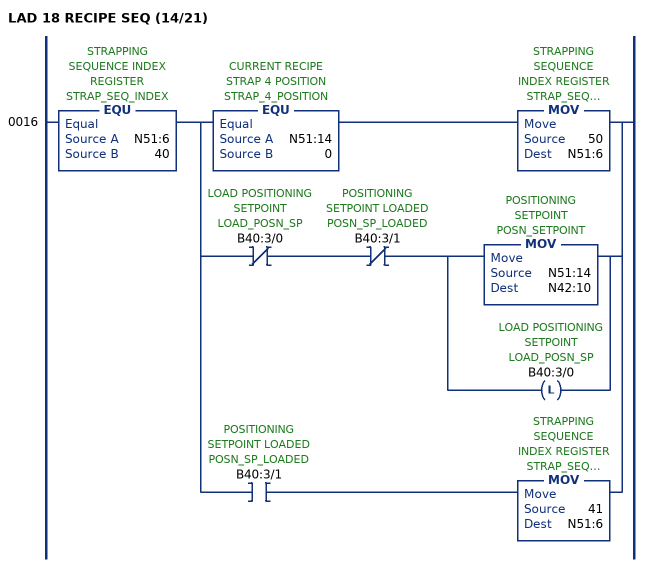
% Rung: 16 %
SOR EQU N51:6 40 BST EQU N51:14 0 MOV 50 N51:6 NXB XIO B40:3/0 XIO B40:3/1 BST MOV N51:14 N42:10 NXB OTL B40:3/0 BND NXB XIC B40:3/1 MOV 41 N51:6 BND EOR
%   N51:6  STRAP_SEQ_INDEX  "STRAPPING SEQUENCE INDEX REGISTER" %
%   N51:14  STRAP_4_POSITION  "CURRENT RECIPE STRAP 4 POSITION" %
%   B40:3/0  LOAD_POSN_SP  "LOAD POSITIONING SETPOINT" %
%   B40:3/1  POSN_SP_LOADED  "POSITIONING SETPOINT LOADED" %
%   N42:10  POSN_SETPOINT  "POSITIONING SETPOINT" %

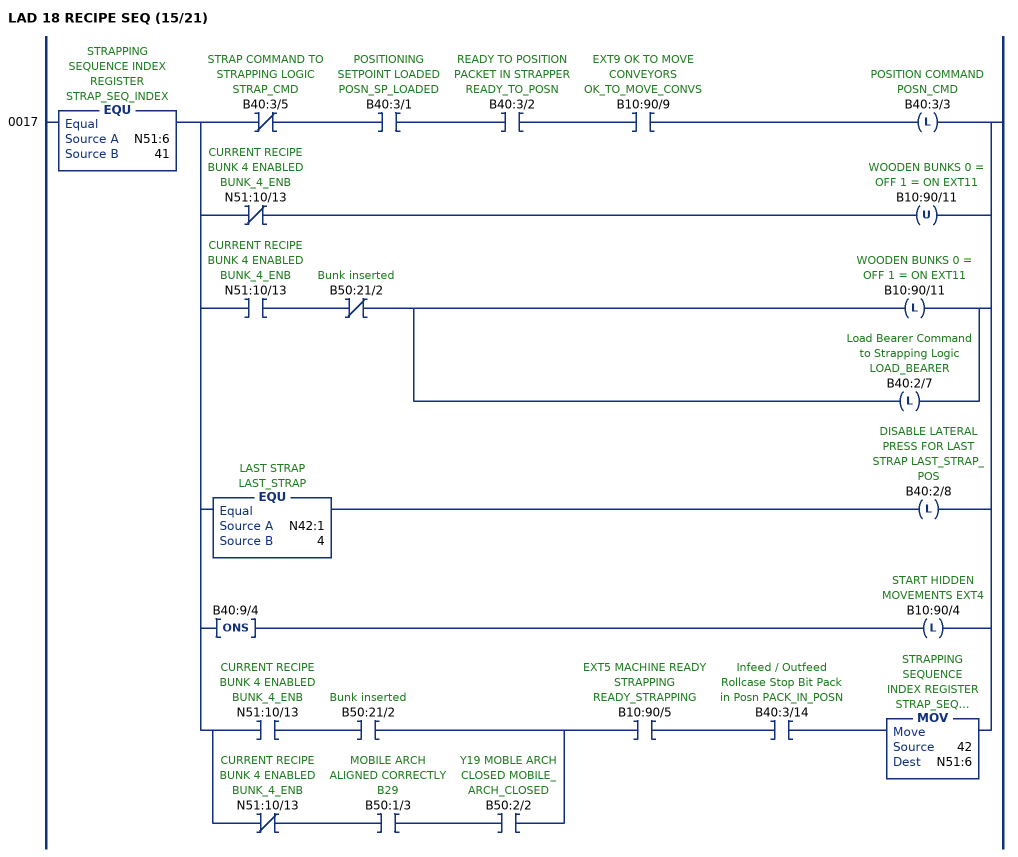
% Rung: 17 %
SOR EQU N51:6 41 BST XIO B40:3/5 XIC B40:3/1 XIC B40:3/2 XIC B10:90/9 OTL B40:3/3 NXB XIO N51:10/13 OTU B10:90/11 NXB XIC N51:10/13 XIO B50:21/2 BST OTL B10:90/11 NXB OTL B40:2/7 BND NXB EQU N42:1 4 OTL B40:2/8 NXB ONS B40:9/4 OTL B10:90/4 NXB BST XIC N51:10/13 XIC B50:21/2 NXB XIO N51:10/13 XIC B50:1/3 XIC B50:2/2 BND XIC B10:90/5 XIC B40:3/14 MOV 42 N51:6 BND EOR
%   N51:6  STRAP_SEQ_INDEX  "STRAPPING SEQUENCE INDEX REGISTER" %
%   B40:3/5  STRAP_CMD  "STRAP COMMAND TO STRAPPING LOGIC" %
%   B40:3/1  POSN_SP_LOADED  "POSITIONING SETPOINT LOADED" %
%   B40:3/2  READY_TO_POSN  "READY TO POSITION PACKET IN STRAPPER" %
%   B10:90/9  OK_TO_MOVE_CONVS  "EXT9 OK TO MOVE CONVEYORS" %
%   B40:3/3  POSN_CMD  "POSITION COMMAND" %
%   N51:10/13  BUNK_4_ENB  "CURRENT RECIPE BUNK 4 ENABLED" %
%   B10:90/11  EXT11  "WOODEN BUNKS 0 = OFF 1 = ON" %
%   B50:21/2  "Bunk inserted" %
%   B40:2/7  LOAD_BEARER  "Load Bearer Command to Strapping Logic" %
%   N42:1  LAST_STRAP  "LAST STRAP" %
%   B40:2/8  LAST_STRAP_POS  "DISABLE LATERAL PRESS FOR LAST STRAP" %
%   B10:90/4  EXT4  "START HIDDEN MOVEMENTS" %
%   B50:1/3  B29  "MOBILE ARCH ALIGNED CORRECTLY" %
%   B50:2/2  MOBILE_ARCH_CLOSED  "Y19 MOBLE ARCH CLOSED" %
%   B10:90/5  READY_STRAPPING  "EXT5 MACHINE READY STRAPPING" %
%   B40:3/14  PACK_IN_POSN  "Infeed / Outfeed Rollcase Stop Bit Pack in Posn" %

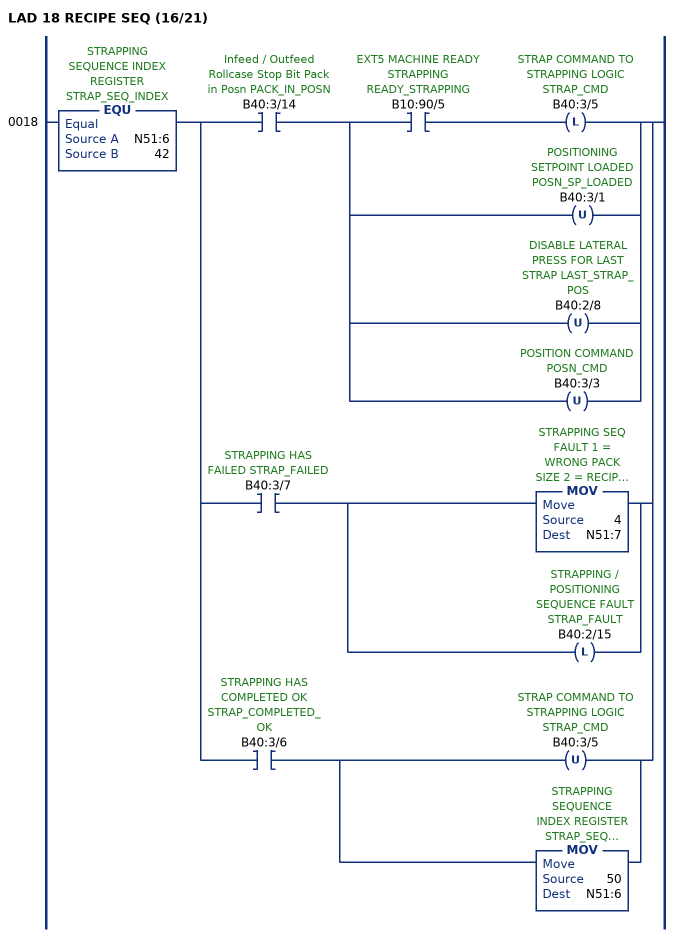
% Rung: 18 %
SOR EQU N51:6 42 BST XIC B40:3/14 BST XIC B10:90/5 OTL B40:3/5 NXB OTU B40:3/1 NXB OTU B40:2/8 NXB OTU B40:3/3 BND NXB XIC B40:3/7 BST MOV 4 N51:7 NXB OTL B40:2/15 BND NXB XIC B40:3/6 BST OTU B40:3/5 NXB MOV 50 N51:6 BND BND EOR
%   N51:6  STRAP_SEQ_INDEX  "STRAPPING SEQUENCE INDEX REGISTER" %
%   B40:3/14  PACK_IN_POSN  "Infeed / Outfeed Rollcase Stop Bit Pack in Posn" %
%   B10:90/5  READY_STRAPPING  "EXT5 MACHINE READY STRAPPING" %
%   B40:3/5  STRAP_CMD  "STRAP COMMAND TO STRAPPING LOGIC" %
%   B40:3/1  POSN_SP_LOADED  "POSITIONING SETPOINT LOADED" %
%   B40:2/8  LAST_STRAP_POS  "DISABLE LATERAL PRESS FOR LAST STRAP" %
%   B40:3/3  POSN_CMD  "POSITION COMMAND" %
%   B40:3/7  STRAP_FAILED  "STRAPPING HAS FAILED" %
%   N51:7  STRAP_SEQ_FLT  "STRAPPING SEQ FAULT 1 = WRONG PACK SIZE 2 = RECIPE FAULT 3 = POSNING FAULT 4 = STRAPPING FAULT" %
%   B40:2/15  STRAP_FAULT  "STRAPPING / POSITIONING SEQUENCE FAULT" %
%   B40:3/6  STRAP_COMPLETED_OK  "STRAPPING HAS COMPLETED OK" %

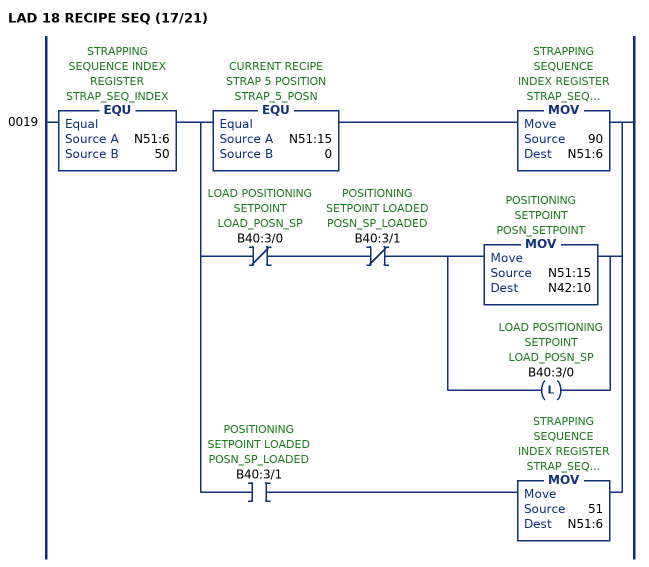
% Rung: 19 %
SOR EQU N51:6 50 BST EQU N51:15 0 MOV 90 N51:6 NXB XIO B40:3/0 XIO B40:3/1 BST MOV N51:15 N42:10 NXB OTL B40:3/0 BND NXB XIC B40:3/1 MOV 51 N51:6 BND EOR
%   N51:6  STRAP_SEQ_INDEX  "STRAPPING SEQUENCE INDEX REGISTER" %
%   N51:15  STRAP_5_POSN  "CURRENT RECIPE STRAP 5 POSITION" %
%   B40:3/0  LOAD_POSN_SP  "LOAD POSITIONING SETPOINT" %
%   B40:3/1  POSN_SP_LOADED  "POSITIONING SETPOINT LOADED" %
%   N42:10  POSN_SETPOINT  "POSITIONING SETPOINT" %

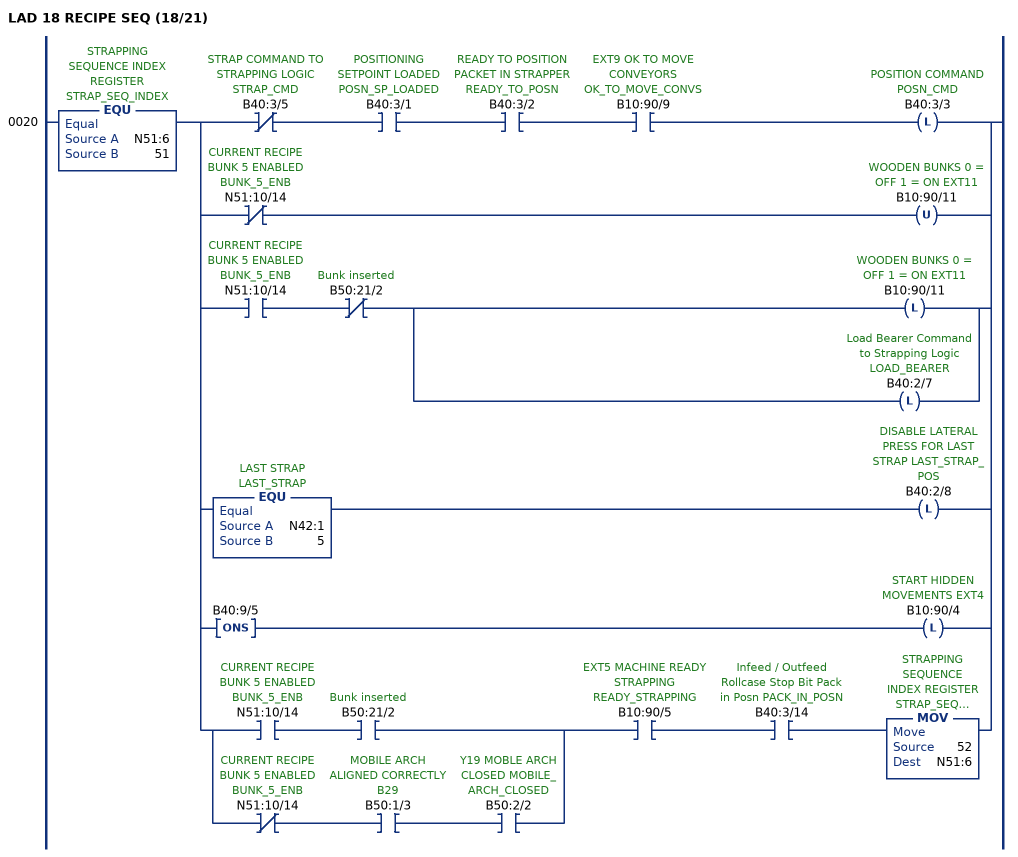
% Rung: 20 %
SOR EQU N51:6 51 BST XIO B40:3/5 XIC B40:3/1 XIC B40:3/2 XIC B10:90/9 OTL B40:3/3 NXB XIO N51:10/14 OTU B10:90/11 NXB XIC N51:10/14 XIO B50:21/2 BST OTL B10:90/11 NXB OTL B40:2/7 BND NXB EQU N42:1 5 OTL B40:2/8 NXB ONS B40:9/5 OTL B10:90/4 NXB BST XIC N51:10/14 XIC B50:21/2 NXB XIO N51:10/14 XIC B50:1/3 XIC B50:2/2 BND XIC B10:90/5 XIC B40:3/14 MOV 52 N51:6 BND EOR
%   N51:6  STRAP_SEQ_INDEX  "STRAPPING SEQUENCE INDEX REGISTER" %
%   B40:3/5  STRAP_CMD  "STRAP COMMAND TO STRAPPING LOGIC" %
%   B40:3/1  POSN_SP_LOADED  "POSITIONING SETPOINT LOADED" %
%   B40:3/2  READY_TO_POSN  "READY TO POSITION PACKET IN STRAPPER" %
%   B10:90/9  OK_TO_MOVE_CONVS  "EXT9 OK TO MOVE CONVEYORS" %
%   B40:3/3  POSN_CMD  "POSITION COMMAND" %
%   N51:10/14  BUNK_5_ENB  "CURRENT RECIPE BUNK 5 ENABLED" %
%   B10:90/11  EXT11  "WOODEN BUNKS 0 = OFF 1 = ON" %
%   B50:21/2  "Bunk inserted" %
%   B40:2/7  LOAD_BEARER  "Load Bearer Command to Strapping Logic" %
%   N42:1  LAST_STRAP  "LAST STRAP" %
%   B40:2/8  LAST_STRAP_POS  "DISABLE LATERAL PRESS FOR LAST STRAP" %
%   B10:90/4  EXT4  "START HIDDEN MOVEMENTS" %
%   B50:1/3  B29  "MOBILE ARCH ALIGNED CORRECTLY" %
%   B50:2/2  MOBILE_ARCH_CLOSED  "Y19 MOBLE ARCH CLOSED" %
%   B10:90/5  READY_STRAPPING  "EXT5 MACHINE READY STRAPPING" %
%   B40:3/14  PACK_IN_POSN  "Infeed / Outfeed Rollcase Stop Bit Pack in Posn" %

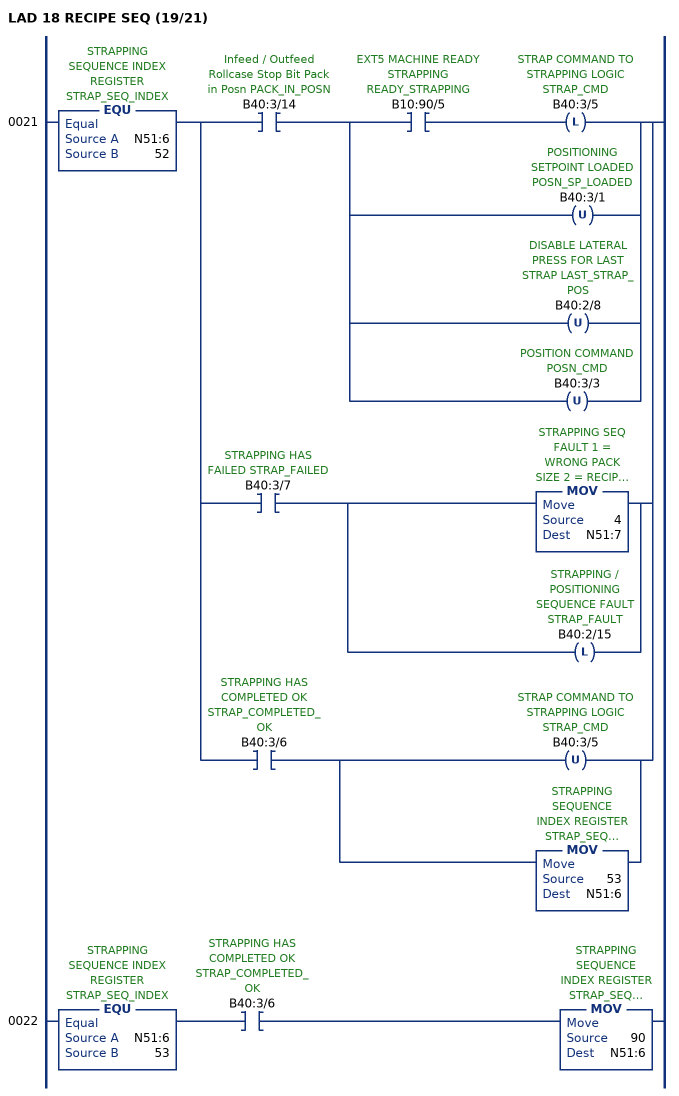
% Rung: 21 %
SOR EQU N51:6 52 BST XIC B40:3/14 BST XIC B10:90/5 OTL B40:3/5 NXB OTU B40:3/1 NXB OTU B40:2/8 NXB OTU B40:3/3 BND NXB XIC B40:3/7 BST MOV 4 N51:7 NXB OTL B40:2/15 BND NXB XIC B40:3/6 BST OTU B40:3/5 NXB MOV 53 N51:6 BND BND EOR
%   N51:6  STRAP_SEQ_INDEX  "STRAPPING SEQUENCE INDEX REGISTER" %
%   B40:3/14  PACK_IN_POSN  "Infeed / Outfeed Rollcase Stop Bit Pack in Posn" %
%   B10:90/5  READY_STRAPPING  "EXT5 MACHINE READY STRAPPING" %
%   B40:3/5  STRAP_CMD  "STRAP COMMAND TO STRAPPING LOGIC" %
%   B40:3/1  POSN_SP_LOADED  "POSITIONING SETPOINT LOADED" %
%   B40:2/8  LAST_STRAP_POS  "DISABLE LATERAL PRESS FOR LAST STRAP" %
%   B40:3/3  POSN_CMD  "POSITION COMMAND" %
%   B40:3/7  STRAP_FAILED  "STRAPPING HAS FAILED" %
%   N51:7  STRAP_SEQ_FLT  "STRAPPING SEQ FAULT 1 = WRONG PACK SIZE 2 = RECIPE FAULT 3 = POSNING FAULT 4 = STRAPPING FAULT" %
%   B40:2/15  STRAP_FAULT  "STRAPPING / POSITIONING SEQUENCE FAULT" %
%   B40:3/6  STRAP_COMPLETED_OK  "STRAPPING HAS COMPLETED OK" %
% Rung: 22 %
SOR EQU N51:6 53 XIC B40:3/6 MOV 90 N51:6 EOR
%   N51:6  STRAP_SEQ_INDEX  "STRAPPING SEQUENCE INDEX REGISTER" %
%   B40:3/6  STRAP_COMPLETED_OK  "STRAPPING HAS COMPLETED OK" %

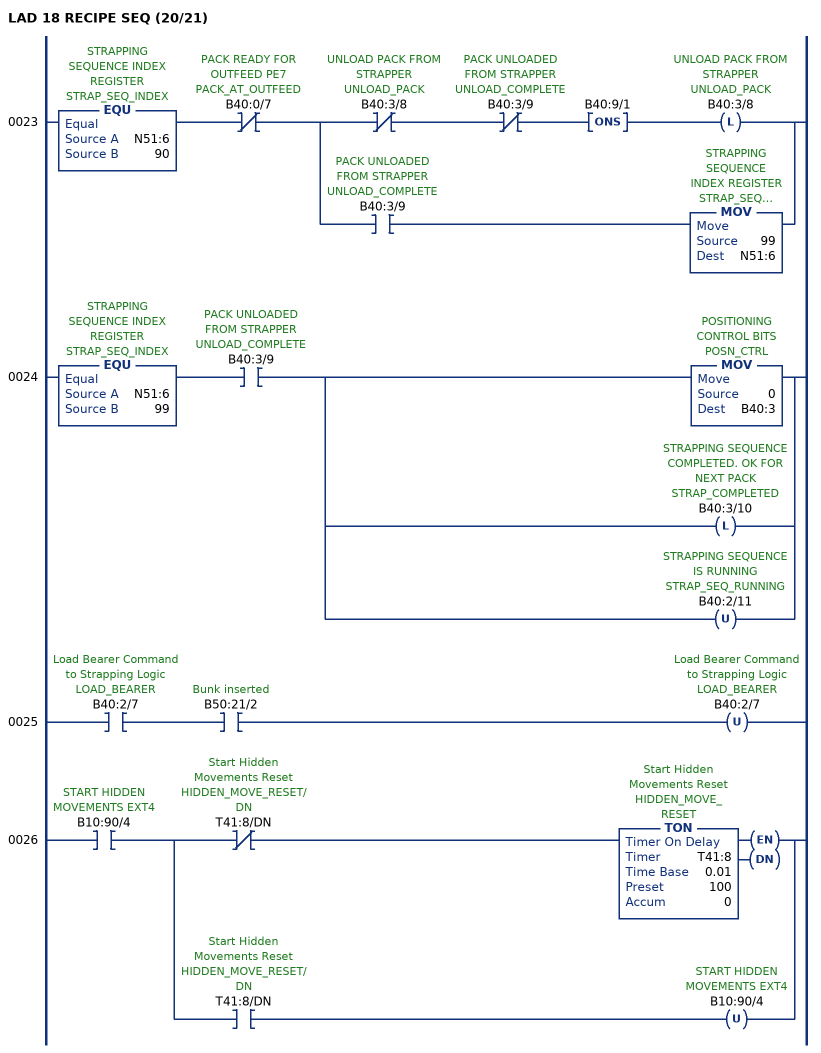
% Rung: 23 %
SOR EQU N51:6 90 XIO B40:0/7 BST XIO B40:3/8 XIO B40:3/9 ONS B40:9/1 OTL B40:3/8 NXB XIC B40:3/9 MOV 99 N51:6 BND EOR
%   N51:6  STRAP_SEQ_INDEX  "STRAPPING SEQUENCE INDEX REGISTER" %
%   B40:0/7  PACK_AT_OUTFEED  "PACK READY FOR OUTFEED PE7" %
%   B40:3/8  UNLOAD_PACK  "UNLOAD PACK FROM STRAPPER" %
%   B40:3/9  UNLOAD_COMPLETE  "PACK UNLOADED FROM STRAPPER" %
% Rung: 24 %
SOR EQU N51:6 99 XIC B40:3/9 BST MOV 0 B40:3 NXB OTL B40:3/10 NXB OTU B40:2/11 BND EOR
%   N51:6  STRAP_SEQ_INDEX  "STRAPPING SEQUENCE INDEX REGISTER" %
%   B40:3/9  UNLOAD_COMPLETE  "PACK UNLOADED FROM STRAPPER" %
%   B40:3  POSN_CTRL  "POSITIONING CONTROL BITS" %
%   B40:3/10  STRAP_COMPLETED  "STRAPPING SEQUENCE COMPLETED. OK FOR NEXT PACK" %
%   B40:2/11  STRAP_SEQ_RUNNING  "STRAPPING SEQUENCE IS RUNNING" %
% Rung: 25 %
SOR XIC B40:2/7 XIC B50:21/2 OTU B40:2/7 EOR
%   B40:2/7  LOAD_BEARER  "Load Bearer Command to Strapping Logic" %
%   B50:21/2  "Bunk inserted" %
% Rung: 26 %
SOR XIC B10:90/4 BST XIO T41:8/DN TON T41:8 0.01 100 0 NXB XIC T41:8/DN OTU B10:90/4 BND EOR
%   B10:90/4  EXT4  "START HIDDEN MOVEMENTS" %
%   T41:8  HIDDEN_MOVE_RESET  "Start Hidden Movements Reset" %

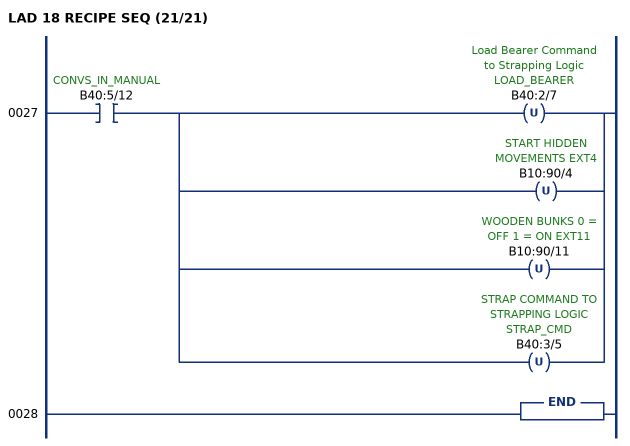
% Rung: 27 %
SOR XIC B40:5/12 BST OTU B40:2/7 NXB OTU B10:90/4 NXB OTU B10:90/11 NXB OTU B40:3/5 BND EOR
%   B40:5/12  CONVS_IN_MANUAL %
%   B40:2/7  LOAD_BEARER  "Load Bearer Command to Strapping Logic" %
%   B10:90/4  EXT4  "START HIDDEN MOVEMENTS" %
%   B10:90/11  EXT11  "WOODEN BUNKS 0 = OFF 1 = ON" %
%   B40:3/5  STRAP_CMD  "STRAP COMMAND TO STRAPPING LOGIC" %
% Rung: 28 %
SOR END EOR

OTHER DOCUMENTED ADDRESSES
  B1:0  "NOEM"
  B3:1/0  "Avl_Pres_vertical"
  B3:1/5  Y23  "Y23"
  B3:1/6  "Avl_Pres_lateral"
  B3:2/3  "IPWR"
  B3:2/4  "Par"
  B3:2/6  "Check_control_motor_ brake"
  B3:14/5  "High_pressure"
  B3:26  MPV  "MPV"
  B3:27  MPL  "MPL"
  B3:28  "FIX_FORCE_V_P"
  B3:29  I  "FIX_FORCE_L_P"
  B10:2/2  "H4"
  B10:2/3  "H5"
  B10:2/4  "EXT25"
  B10:2/5  "EXT26"
  B10:2/6  "EXT27"
  B10:2/7  "EXT28"
  B10:15/0  "OP_V_F_PRESS"
  B10:17/0  "Pack_Large"
  B10:18/0  "C_lpress_FIX_press"
  B10:19/0  "B_vpress_FIX_press"
  B10:33/5  F6  "F6-KEY"
  B10:90/0  "EXT0"
  B10:90/1  "EXT1"
  B10:90/2  "EXT2"
  B10:90/3  "EXT3"
  B10:90/7  "EXT7"
  B10:90/14  "EXT14"
  B10:90/15  "EXT15"
  B10:91/0  "EXT16"
  B10:91/1  "EXT17"
  B10:91/2  "EXT18"
  B10:91/3  "EXT19"
  B10:91/8  "EXT24"
  B10:100/6  "G_Corner"
  B10:100/7  "B_vpress_FIX_pres"
  B10:100/8  "C_lpress_FIX_pres"
  B10:100/9  "Pack_small"
  B20:0/2  "B3"
  B20:200/1  "E2"
  B40:0/12  PACK_STORAGE_PE_2  "Pack Index Point 3"
  B40:2/12  STRAP_SEQ_COMPLETE  "STRAPPING SEQUENCE IS COMPLETE"
  B40:3/4  PACK_POSNED  "PACK IS POSITIONED IN STRAPPER"
  B40:4  POSN_CTRL_2  "Position Control Bits Word 2"
  B40:4/6  LOAD_BEARER_PULSE  "Load Bearer Pulse To Strapping Logic"
  B40:5  DECK_CTRL  "Infeed and Outfeed Deck Control Bits"
  B40:5/14  IFEED_MAN_LOWER  "Infeed Deck Lower Manual"
  B40:6/1  OFFED_LOWER_MAN  "Outfeed Deck Lower Manual"
  B40:9  ONE_SHOTS
  B40:10/2  PACK_AT_INDEX_2  "PACK AT INDEX POINT 2"
  B50:0/6  "E25"
  B50:0/7  "E26"
  B50:0/11  "SS7"
  B50:0/12  "SS8"
  B50:0/13  "SS9"
  B50:1/10  "E43"
  B50:1/11  "E44"
  B50:1/12  "E45"
  B50:3/3  "X43"
  B50:3/4  "X44"
  B50:3/5  "X44_1"
  B50:3/6  "X44_2"
  B50:3/7  "X44_3"
  B50:3/8  "X44_4"
  B50:3/9  "X43_1"
  B50:3/10  "X43_2"
  B50:4/1  "Ok_mag_E"
  B50:4/2  "Ok_mag_F"
  B50:7/0  "X29_1"
  B50:7/1  "X29_2"
  B50:7/4  "X30_3"
  B50:7/5  "X30_4"
  B50:7/8  "X31_3"
  B50:7/9  "X32_1"
  B50:7/10  "X32_2"
  B50:7/11  "X32_3"
  B50:11/5  "Mag_allinead2"
  B50:14/8  "Mag_D_empty"
  B50:14/9  "Mag_E_empty"
  B50:14/10  "Mag_F_empty"
  B50:30/0  "Bunk A=1140 mm"
  B50:31/0  "Bunk B=1140 mm"
  B50:32/0  "Bunk C=1140 mm"
  B50:33/0  "Bunk D=1140 mm"
  B50:34/0  "Bunk E=1140 mm"
  B50:35/0  "Bunk F=1140 mm"
  B50:80/1  "E34"
  B50:80/3  "E36"
  B50:80/4  "E37"
  B50:80/7  "E38"
  F8:5  SPEED_CH_SP_3  "Speed Change Setpoint 3 (0 - 100%)"
  HSC:0.5  HSC_ACC  "High Speed Counter Accumulator"
  I:0.0/0  ENCODER_A  "ENCODER A COUNT"
  I:0.0/1  ENCODER_B  "ENCODER B COUNT"
  I:0.0/2  ENCODER_Z  "ENCODER Z COUNT (UNUSED)"
  I:3.0/6  "START HIDDEN MOVEMENTS"
  I:3.0/7  "START STRAPPING PRESSING"
  I:3.0/8  "WOODEN BUNKS 0 = OFF 1 = ON"
  I:3.0/9  "STRAPPING 0 = OFF 1 = ON"
  I:3.0/10  "PRESS VERTICAL 0 = OFF 1 = ON"
  I:3.0/11  "PRESS LATERAL 0 = OFF 1 = ON"
  I:4.0/9  "CYCLE START HIDDEN MOVEMENTS WOODEN BUNK STORE 1"
  I:4.0/10  "CYCLE START HIDDEN MOVEMENTS WOODEN BUNK STORE 2"
  I:4.0/11  "CYCLE START HIDDEN MOVEMENTS WOODEN BUNK STORE 3"
  L9:0  ENCODER_RAW_ACC  "Raw Accumulator Counts from Encoder Input"
  L9:1  ENCODER_RAW_MIN  "Minimum Raw Input From Encoder"
  L9:2  "Maximum Raw Input From Encoder"
  N7:2  ACTUAL_POSN  "Encoder Actual Position (Scaled)"
  N7:7  ENCODER_SCL_MIN  "Encoder Scaled Minimum (mm + 2DP)"
  N7:8  ENCODER_SCL_MAX  "Encoder Scaled Maximum (mm + 2DP)"
  N9:24  "PAG"
  N42:0  INDEX_DEST  "PACK INDEX DESTINATION"
  N51:1  CURRENT_SCREEN  "CURRENT SCREEN BEING DISPLAYED"
  N51:20  RECIPE_1  "RECIPE 1"
  N51:26  REC_1_BUNK_MAG  "Recipe 1 Bunk Magazine"
  N51:30  RECIPE_2  "RECIPE 2"
  N51:36  REC_2_BUNK_MAG  "Recipe 2 Bunk Magazine"
  N51:40  RECIPE_3  "RECIPE 3"
  N51:46  REC_3_BUNK_MAG  "Recipe 3 Bunk Magazine"
  N51:50  RECIPE_4  "RECIPE 4"
  N51:56  REC_4_BUNK_MAG  "Recipe 4 Bunk Magazine"
  N51:60  RECIPE_5  "RECIPE 5"
  N51:66  REC_5_BUNK_MAG  "Recipe 5 Bunk Magazine"
  N51:70  RECIPE_6  "RECIPE 6"
  N51:76  REC_6_BUNK_MAG  "Recipe 6 Bunk Magazine"
  N51:80  RECIPE_7  "RECIPE 7"
  N51:90  RECIPE_8  "RECIPE 8"
  N51:100  RECIPE_9  "RECIPE 9"
  N51:110  RECIPE_10  "RECIPE 10"
  N51:120  RECIPE_11  "RECIPE 11"
  N51:130  RECIPE_12  "RECIPE 12"
  N51:140  RECIPE_13  "RECIPE 14"
  N51:170  NEXT_RECIPE_NAME  "NEXT RECIPE NAME"
  O:1.2  OUTFEED_VSD_RAW_OUT  "Outfeed Rollcase VSD Raw Speed Reference Out"
  O:7.0/2  "CYCLE END EXT 6"
  ST52:0  CURR_REC_NAME  "CURRENT RECIPE NAME"
  T4:11  "TM-"
  T4:20  "TV-"
  T4:25  "TAA-"
  T4:26  "TAB-"
  T4:27  "TAC-"
  T4:28  "TAD-"
  T4:29  "TAE-"
  TB  "q"

COMMENTS NOT ATTACHED TO A CURRENT RUNG
  B3:4/2: ******************************************************WARNING************************************************************
    THIS COMPUTER PROGRAM IS PROTECTED BY COPYRIGHTLAW AND  INTERNATIONALTREATIES.UNAUTHORIZED
     REPRODUCTION OR DISTRIBUTION OF THIS PROGRAM  OR ANY PORTION  OF IT,MAY RESULT IN SEVERE CIVIL
    AND  CRIMINAL PENALTIES ,AND WILL BE PROSECUTED TO THE MAXIMUM EXTENE POSSIBLE  UNDER THE LAW **************************************************************************************************************************
    HEAD MOTION ON FAST SPEED TILL E 10 THEN STOP
    DEPPRESSING AND THEN PRESSING AGAIN NTHE FUNCTION KEY, THE MOVEMENT STARTS AGAIN ON SLOW SPEED
  B3:8/6: RESET AT THE END OF CYCLE
  B3:10/5: RESET
  B3:2/3: HEAD STROKE - INVERTER SUPPLY AUX
  B3:1/9: By pass oil central unit
  N7:30/5: WELDING BLADE TOO COLD
  N7:31/13: RESET MACHINE NOT POSSIBLE
  N7:32/1: TIMEOUT STRAP FEEDING
  N7:32/2: Check contactors brake motor
  N7:32/8: STRAP FEEDING FAILURE
  N7:32/9: STRAP TAKE-UP FAILURE
  O:3.0/0: IMAGE OUTPUT / ******************************************************WARNING************************************************************
    THIS COMPUTER PROGRAM IS PROTECTED BY COPYRIGHTLAW AND  INTERNATIONALTREATIES.UNAUTHORIZED
     REPRODUCTION OR DISTRIBUTION OF THIS PROGRAM  OR ANY PORTION  OF IT,MAY RESULT IN SEVERE CIVIL
    AND  CRIMINAL PENALTIES ,AND WILL BE PROSECUTED TO THE MAXIMUM EXTENE POSSIBLE  UNDER THE LAW **************************************************************************************************************************
  N7:32/0: STRAP UNLOCKED
  B50:4/2: Magazine F
  B50:4/1: Magazine E
  N7:32/6: MACHINE RESET IMPOSSIBLE
  N7:33/2: STRAP TAKE-UP FAILURE
  B3:1/10: Vertical press high pressure
  N7:61: --------------------------------------------------------------------------------------------------Monitor inputs------------------------------------------------------------------------------------------------
  N7:30/4: Safety Arch
  N7:30/6: Welding blade not ready to work
  N7:31/1: Cams timeout
  N7:32/7: MAGASINE A EMPTY
  N7:32/13: Magazine  door opened
  N7:33/3: TIMEOUT MOVEMENT BUNK PUSHER FORWARD
  N7:33/4: TIMEOUT RIGHT PUSHER CORNER
  N7:33/5: TIMEOUT LEFT PUSHER CORNER
  N7:33/6: RIGHT MAGAZINE CORNERS EMPTY
  B3:2/4: Press force during strapping
  N11:0/9: Key   F3   page up
  N11:0/11: Key F4 Pag down
  N7:31/6: MACHINE RESET IMPOSSIBLE
  N7:31/10: TIMEOUT MOVIMENT HEAD DOWN
  N7:31/11: I001 - STRAP FINISHED
  B10:104/2: AUTOMATIC REGULAR
  B10:92/2: EXT 10 Fault machine
  B3:1/5: BY - PASS OIL UNIT
  N42:0: Determine how many packs are on deck to index
    0 = Deck Full, can't index
    10 = 1 Pack at Index Point 2, Load to Index Point 1
    20 = 1 Pack at Index Point 3, Load to Index Point 2
    30 = Pack on Rollcase or in Strapper, Load to Index Point 3
    40 = Deck Empty - Load to Rollcase
  B10:103/1: REQUEST CYCLE STRAPPING

DATA TABLE (non-zero values as saved)
DATA B3
% B3:0 % 0X0007 0X0000 0X004C 0X0000 0X0000 0X0000 0X0000 0X0000 0X0000 0X0000
% B3:20 % 0X01A7 0X0000 0X0000 0X0000 0X0000 0X0000 0X0032 0X0032 0X0000 0X0000
DATA T4
% .PRE .ACC %
% T4:0 % 650 0
% T4:1 % 250 0
% T4:2 % 500 0
% T4:3 % 400 0
% T4:4 % 50 0
% T4:5 % 250 0
% T4:6 % 100 0
% T4:7 % 100 0
% T4:8 % 100 0
% T4:9 % 6000 0
% T4:10 % 50 0
% T4:12 % 40 0
% T4:13 % 6 0
% T4:14 % 130 0
% T4:15 % 20 0
% T4:17 % 500 0
% T4:18 % 300 0
% T4:19 % 6000 0
% T4:21 % 600 0
% T4:22 % 180 0
% T4:23 % 25 25
% T4:24 % 400 136
% T4:30 % 350 0
% T4:31 % 350 0
% T4:32 % 600 0
% T4:33 % 600 0
% T4:34 % 600 0
% T4:35 % 350 0
% T4:36 % 50 0
% T4:37 % 700 0
% T4:38 % 700 0
% T4:39 % 90 0
% T4:40 % 6000 0
% T4:41 % 200 0
% T4:42 % 50 0
% T4:43 % 60 60
% T4:44 % 200 0
% T4:45 % 800 0
% T4:46 % 40 0
% T4:47 % 900 0
% T4:48 % 100 0
% T4:49 % 900 0
% T4:51 % 900 0
DATA N7
% N7:0 % 3 0 0 0 0 25 25 0 0 0
% N7:10 % 4 0 30001 0 0 0 0 0 0 0
% N7:20 % 0 0 0 0 30001 0 0 0 0 0
% N7:30 % 1 0 0 0 0 0 0 0 0 0
% N7:40 % 90 90 90 90 90 90 90 90 90 90
% N7:50 % 90 90 90 90 90 0 0 0 0 0
% N7:60 % 0 -14535 -29128 38 0 16426 3 0
DATA F8
% F8:0 % -60.912 0 0 -300 -150
% F8:5 % 0 300 150 0
DATA N9
% N9:0 % 0 0 1 30 0 0 0 0 0 0
% N9:10 % 1 0 1
DATA B10
% B10:0 % 0X0004 0X0003 0X0000 0X0000 0X0000 0X0000 0X0000 0X0000 0X0000 0X0000
% B10:10 % 0X0000 0X0001 0X0001 0X0000 0X0000 0X0000 0X0000 0X0000 0X0000 0X0000
% B10:40 % 0X0004 0X0000 0X0000 0X0000 0X0000 0X0000 0X0000 0X0000 0X0000 0X0000
% B10:90 % 0X3200 0X0030 0X0000 0X0000 0X0000 0X0008 0X0000 0X0000 0X0000 0X0000
% B10:100 % 0X0000 0X0001 0X0000 0X0000 0X0000 0X0000
DATA N11
% N11:0 % 7684 24576 2
DATA L12
% L12:0 % 2648 52 0 0 0
% L12:10 % 0 0 15803 0 32767
% L12:15 % 52
DATA B20
% B20:0 % 0X0028 0X0000 0X0000 0X000F 0X0000 0X0000 0X0000 0X0000 0X0000 0X0000
% B20:10 % 0X0000 0X0004 0X0000 0X0000 0X0000 0X0000 0X0000 0X0000 0X0000 0X0000
% B20:20 % 0X0000 0X0040 0X0000 0X0000 0X0000 0X0000 0X0000 0X0000 0X0000 0X0000
% B20:90 % 0X0005 0X0000 0X0000 0X0000 0X0001 0X0000 0X0064 0X0000 0X0000 0X0000
% B20:100 % 0X000E
DATA B35
% B35:0 % 0X0004 0X0000 0X0000 0X0000 0X0000 0X0001 0X0000 0X0000 0X0000
DATA B40
% B40:0 % 0X0000 0X000A 0X0000 0X0000 0X0031 0X1000 0X0000 0X0000 0X0000 0X0000
DATA T41
% .PRE .ACC %
% T41:0 % 20 0
% T41:1 % 1000 0
% T41:2 % 50 0
% T41:3 % 900 0
% T41:4 % 2000 0
% T41:5 % 50 0
% T41:6 % 50 0
% T41:7 % 300 0
% T41:8 % 100 0
% T41:9 % 100 0
% T41:10 % 800 0
% T41:11 % 600 0
% T41:12 % 20 0
% T41:13 % 500 500
DATA N42
% N42:0 % 0 3 0 0 0 0 0 0 0 0
% N42:10 % 0 764 0 0 0 0 0 0 0 0
% N42:20 % 8192 0 0 0 0 0 0 0 0 0
% N42:90 % 100 50 25 0 0 100 0 16383 0 0
DATA B50
% B50:0 % 0X3F55 0X03B1 0X0040 0X0209 0X0000 0X0000 0X0000 0X0240 0X0000 0X0000
% B50:10 % 0X0000 0X0029 0X0080 0X0000 0X0000 0X0004 0X0000 0X0000 0X0000 0X0000
DATA N51
% N51:0 % 4 0 50 0 0 0 0 2 0 0
% N51:10 % 7170 300 1710 1710 0 0 1 0 0 0
% N51:20 % 21506 305 835 835 835 835 1 0 0 0
% N51:30 % 21506 300 835 835 835 835 2 0 0 0
% N51:40 % 31746 300 850 850 850 850 3 0 0 0
% N51:50 % 7170 300 1710 1710 0 0 1 0 0 0
% N51:60 % 7170 300 1710 1710 0 0 2 0 0 0
% N51:70 % 7170 300 1710 1710 0 0 3 0 0 0
% N51:80 % 7169 300 1200 1200 0 0 1 0 0 0
% N51:90 % 7169 300 1200 1200 0 0 2 0 0 0
% N51:100 % 7169 300 1200 1200 0 0 3 0 0 0
% N51:110 % 3073 300 2410 0 0 0 1 0 0 0
% N51:120 % 3073 300 2410 0 0 0 2 0 0 0
% N51:130 % 3073 300 2410 0 0 0 3 0 0 0
% N51:150 % 4 0 0 0 0 0 0 0 0 0
% N51:160 % 7170 300 1710 1710 0 0 1 0 0 0
DATA N52
% N52:0 % 12865 0 0 0 0 0 0 0 0 0
% N52:10 % 12609 0 0 0 0 0 0 0 0 0
% N52:20 % 12610 0 0 0 0 0 0 0 0 0
% N52:30 % 12611 0 0 0 0 0 0 0 0 0
% N52:40 % 12865 0 0 0 0 0 0 0 0 0
% N52:50 % 12866 0 0 0 0 0 0 0 0 0
% N52:60 % 12867 0 0 0 0 0 0 0 0 0
% N52:70 % 13121 0 0 0 0 0 0 0 0 0
% N52:80 % 13122 0 0 0 0 0 0 0 0 0
% N52:90 % 13123 0 0 0 0 0 0 0 0 0
% N52:100 % 13377 0 0 0 0 0 0 0 0 0
% N52:150 % 12865 0 0 0 0 0 0 0 0 0
